// TwinCAT 3 PLC project PLC
// ProgramVersion: 3.1.4026.19
// libraries:
//   SPT Base Types, * (Beckhoff Automation LLC)
//   SPT Components, * (Beckhoff Automation LLC)
//   SPT Diagnostic, * (Beckhoff Automation LLC)
//   SPT EtherCat, * (Beckhoff Automation LLC)
//   SPT Event Logger, * (Beckhoff Automation LLC)
//   SPT Motion Control, * (Beckhoff Automation LLC)
//   SPT Utilities, * (Beckhoff Automation LLC)
//   Tc2_MC2, * (Beckhoff Automation GmbH)
//   Tc2_Standard, * (Beckhoff Automation GmbH)
//   Tc2_System, * (Beckhoff Automation GmbH)
//   Tc3_EventLogger, * (Beckhoff Automation GmbH)
//   Tc3_Module, * (Beckhoff Automation GmbH)
//   Tc3_PackML_V3, * (Beckhoff Automation GmbH)
// project tree:
//   / GlobalTextList.TcGTLO, PlcTask.TcTTO, Visualization Manager.TcVMO (not stored)
//   POUs/ MAIN.TcPOU
//   POUs/Modules/00 Machine/ Machine.TcPOU
//   POUs/Modules/01 Virtual Master/ VirtualMaster.TcPOU
//   POUs/Modules/02 Unwind/ Unwind.TcPOU
//   POUs/Modules/03 Draw/ DrawAxis.TcPOU
//   VISUs/ Visualization.TcVIS
// real-time tasks:
//   TASK PlcTask: cycle T#10ms, priority 20, ADS port 350
// motion (NC):
//   TASK NC-Task 1 SAF: cycle T#2ms, priority 4, ADS port 501
//   TASK NC-Task 1 SVB: cycle T#10ms, priority 8, ADS port 511
//   AXIS Virtual Master (id 1)
//   AXIS Unwind (id 2)
//   AXIS Draw (id 3)
// variable links:
//   PLC/PLC Instance <-> NC-Task 1 SAF/Axes/Draw
//     PlcTask Inputs/MAIN.Machine.Draw.Axis.BasicSlaveAxis._Axis.NcToPlc <-> Outputs/ToPlc
//     PlcTask Outputs/MAIN.Machine.Draw.Axis.BasicSlaveAxis._Axis.PlcToNc <-> Inputs/FromPlc
//   PLC/PLC Instance <-> NC-Task 1 SAF/Axes/Unwind
//     PlcTask Inputs/MAIN.Machine.Unwind.Axis.BasicSlaveAxis._Axis.NcToPlc <-> Outputs/ToPlc
//     PlcTask Outputs/MAIN.Machine.Unwind.Axis.BasicSlaveAxis._Axis.PlcToNc <-> Inputs/FromPlc
//   PLC/PLC Instance <-> NC-Task 1 SAF/Axes/Virtual Master
//     PlcTask Inputs/MAIN.Machine.VirtualMaster.Axis.BasicSlaveAxis._Axis.NcToPlc <-> Outputs/ToPlc
//     PlcTask Outputs/MAIN.Machine.VirtualMaster.Axis.BasicSlaveAxis._Axis.PlcToNc <-> Inputs/FromPlc

CONFIGURATION PLC
    RESOURCE PLC ON TwinCAT3
        TASK PlcTask(INTERVAL := T#10ms, PRIORITY := 20);
        PROGRAM MAIN WITH PlcTask : MAIN;
    END_RESOURCE
END_CONFIGURATION

// ---- POUs/MAIN.TcPOU
PROGRAM MAIN
VAR
	Machine : Machine := (Name := 'Machine');
END_VAR

(*All sample code provided by Beckhoff Automation LLC are for illustrative purposes only and are provided “as is” and without any warranties, express or implied. Actual implementations in applications will vary significantly. Beckhoff Automation LLC shall have no liability for, and does not waive any rights in relation to, any code samples that it provides or the use of such code samples for any purpose.*)

(*
	This code is not a full implementation as there is no use of MC_Reset or other needed code for actual machine use.
	Take note of step 10 in FB_Machine.Initialize, this is where the Axes are assigned to their Master.
	The Unwind Axis makes use of a Gear Ratio in its Coupling.
	There is no code to move the master axis, but it can be jogged from the NC for testing.
*)

// For Debug Only
_AppInfo.KeepOutputsOnBP := TRUE;

//
Machine.CyclicLogic();

END_PROGRAM

// ---- POUs/Modules/00 Machine/Machine.TcPOU
FUNCTION_BLOCK Machine EXTENDS FB_PackML_BaseModule
VAR
	VirtualMaster : VirtualMaster := (Name := 'Virtual Master');
	Unwind		  : Unwind		  := (Name := 'Unwind');
	Draw		  : DrawAxis	  := (Name := 'Draw');
END_VAR

METHOD PUBLIC CyclicLogic
IF NOT _InitComplete THEN
	_InitComplete := Initialize();
	RETURN;
END_IF

SUPER^.CyclicLogic();
END_METHOD

// Automatically enables and disables HMI control based on the PackML mode
METHOD PROTECTED HMIPermissions

// This method is called cyclically by CyclicLogic()
AllowHMIControl(ThisModuleOnly := TRUE);
END_METHOD

METHOD PROTECTED Initialize : BOOL;
Initialize := FALSE;
CASE DescendantSequenceState OF
	0: // Register Submodules
		RegisterSubmodule(VirtualMaster);
		RegisterSubmodule(Unwind);
		RegisterSubmodule(Draw);
		DescendantSequenceState := DescendantSequenceState + 10;

	10: // Assign axis references between Equipment Modules
		Unwind.MasterAxisRef	REF= VirtualMaster.AxisRef;
		Draw.MasterAxisRef		REF= VirtualMaster.AxisRef;
		DescendantSequenceState := DescendantSequenceState + 10;

	20:
		IF SUPER^.Initialize() THEN
			DescendantSequenceState := DescendantSequenceState + 10;
		END_IF

	30:
		Initialize := TRUE;
END_CASE
END_METHOD

END_FUNCTION_BLOCK

// ---- POUs/Modules/01 Virtual Master/VirtualMaster.TcPOU
FUNCTION_BLOCK VirtualMaster EXTENDS FB_PackML_BaseModule
VAR
	Axis : FB_Component_BasicSlaveAxis := (Name := 'Virtual Master Axis');
END_VAR

METHOD PROTECTED Aborting
//Mode is ignored
CASE SequenceState OF
	0:
		// Stop Axis
		Axis.Override := 100;
		IF Axis.Stop() OR Axis.Error THEN // This will also GearOut
			SequenceState := SequenceState + 10;
		END_IF

	10:
		IF Axis.Stopped THEN
			SequenceState := SequenceState + 10;
		END_IF

	20: // Disable Axis
		IF Axis.Disable() THEN
			SequenceState := SequenceState + 10;
		END_IF

	30:
		IF NOT Axis.Enabled THEN
			SequenceState := SequenceState + 10;
		END_IF

	40:
		SUPER^.Aborting();
END_CASE
END_METHOD

PROPERTY AxisRef : REFERENCE TO AXIS_REF
GET
AxisRef REF= Axis.Axis;
END_GET
END_PROPERTY

METHOD PROTECTED Completing
CASE _CurrentMode OF
	E_PMLUnitMode.Production:
		CASE SequenceState OF
			0:
				NoStateTasksToComplete := FALSE;
				IF Axis.Stop() THEN
					SequenceState := SequenceState + 10;
				END_IF

			10:
				IF Axis.Stopped THEN
					SequenceState := SequenceState + 10;
				END_IF

			20:
				StateTasksComplete := TRUE;
		END_CASE

	E_PMLUnitMode.Maintenance, E_PMLUnitMode.Manual:
		;
END_CASE

SUPER^.Completing();
END_METHOD

METHOD PUBLIC CyclicLogic
IF NOT _InitComplete THEN
	_InitComplete := Initialize();
	RETURN;
END_IF

SUPER^.CyclicLogic();
END_METHOD

METHOD PROTECTED Initialize : BOOL;
Initialize := FALSE;
CASE DescendantSequenceState OF
	0:
		RegisterComponent(Axis);
		DescendantSequenceState := DescendantSequenceState + 10;

	10:
		IF SUPER^.Initialize() THEN
			DescendantSequenceState := DescendantSequenceState + 10;
		END_IF

	20:
		Initialize := TRUE;
END_CASE
END_METHOD

METHOD PROTECTED Starting
CASE _CommandedMode OF
	E_PMLUnitMode.Production:
		CASE SequenceState OF
			0:
				NoStateTasksToComplete := FALSE;
				IF Axis.Enable() THEN
					SequenceState := SequenceState + 10;
				END_IF

			10:
				IF Axis.Enabled THEN
					SequenceState := SequenceState + 10;
				END_IF

			20:
				StateTasksComplete := TRUE;
		END_CASE
END_CASE

SUPER^.Starting();
END_METHOD

METHOD PROTECTED Stopping
CASE _CurrentMode OF
	E_PMLUnitMode.Production:
		CASE SequenceState OF
			0:
				NoStateTasksToComplete := FALSE;
				IF Axis.Stop() THEN //This will also GearOut
					SequenceState := SequenceState + 10;
				END_IF

			10:
				IF Axis.Stopped THEN
					SequenceState := SequenceState + 10;
				END_IF

			20:
				StateTasksComplete := TRUE;
		END_CASE
END_CASE

SUPER^.Stopping();
END_METHOD

END_FUNCTION_BLOCK

// ---- POUs/Modules/02 Unwind/Unwind.TcPOU
FUNCTION_BLOCK Unwind EXTENDS FB_PackML_BaseModule
VAR
	Axis	   : FB_Component_BasicSlaveAxis := (Name := 'Unwind Axis');
	_MasterRef : REFERENCE TO AXIS_REF;
END_VAR

METHOD PROTECTED Aborting
//Mode is ignored
CASE SequenceState OF
	0:
		NoStateTasksToComplete := FALSE;

		// Stop Axis
		Axis.Override := 100;
		IF Axis.Stop() OR Axis.Error THEN //This will also GearOut
			SequenceState := SequenceState + 10;
		END_IF

	10:
		IF Axis.Stopped THEN
			SequenceState := SequenceState + 10;
		END_IF

	20: // Disable Axis 
		IF Axis.Disable() THEN
			SequenceState := SequenceState + 10;
		END_IF

	30:
		IF NOT Axis.Enabled THEN
			SequenceState := SequenceState + 10;
		END_IF

	40:
		StateTasksComplete := TRUE;
END_CASE

SUPER^.Aborting();
END_METHOD

PROPERTY AxisRef : REFERENCE TO AXIS_REF
GET
AxisRef REF= Axis.Axis;
END_GET
END_PROPERTY

METHOD PROTECTED Completing
VAR_INST
	StopAxis : BOOL;
END_VAR
CASE _CurrentMode OF
	E_PMLUnitMode.Production:
		CASE SequenceState OF
			0:
				NoStateTasksToComplete := FALSE;
				IF Axis.InGear AND_THEN Axis.Master1.Status.StandStill THEN //Wait for Master Axis to Stop
					StopAxis := TRUE;
				ELSIF NOT Axis.InGear THEN
					StopAxis := TRUE;
				ELSE
					StopAxis := FALSE;
				END_IF

				IF StopAxis AND_THEN Axis.Stop() THEN // This will also GearOut
					SequenceState := SequenceState + 10;
				END_IF

			10:
				IF Axis.Stopped THEN
					SequenceState := SequenceState + 10;
				END_IF

			20:
				StateTasksComplete := TRUE;
		END_CASE

	E_PMLUnitMode.Maintenance, E_PMLUnitMode.Manual:
		;
END_CASE

SUPER^.Completing();
END_METHOD

METHOD PUBLIC CyclicLogic
IF NOT _InitComplete THEN
	_InitComplete := Initialize();
	RETURN;
END_IF

SUPER^.CyclicLogic();
END_METHOD

METHOD PROTECTED Initialize : BOOL;
Initialize := FALSE;
CASE DescendantSequenceState OF
	0:
		RegisterComponent(Axis);
		DescendantSequenceState := DescendantSequenceState + 10;

	10:
		IF SUPER^.Initialize() THEN
			DescendantSequenceState := DescendantSequenceState + 10;
		END_IF

	20:
		Initialize := TRUE;
END_CASE
END_METHOD

PROPERTY MasterAxisRef : REFERENCE TO AXIS_REF
SET
IF __ISVALIDREF(MasterAxisRef) THEN
	_MasterRef REF= MasterAxisRef;
END_IF
END_SET
END_PROPERTY

METHOD PROTECTED Starting
CASE _CommandedMode OF
	E_PMLUnitMode.Production:
		CASE SequenceState OF
			0:
				NoStateTasksToComplete := FALSE;
				IF Axis.Enable() THEN
					SequenceState := SequenceState + 10;
				END_IF

			10:
				IF Axis.Enabled THEN
					SequenceState := SequenceState + 10;
				END_IF

			20:
				Axis.Master1	  REF= _MasterRef;
				Axis.RatioMaster1 := 0.5; //Can be set at anytime and changed while in motion
				IF Axis.GearIn() THEN
					SequenceState := SequenceState + 10;
				END_IF

			30:
				IF Axis.InGear THEN
					SequenceState := SequenceState + 10;
				END_IF

			40:
				StateTasksComplete := TRUE;
		END_CASE
END_CASE

SUPER^.Starting();
END_METHOD

METHOD PROTECTED Stopping
CASE _CurrentMode OF
	E_PMLUnitMode.Production:
		CASE SequenceState OF
			0:
				NoStateTasksToComplete := FALSE;
				IF Axis.Stop() THEN //This will also GearOut
					SequenceState := SequenceState + 10;
				END_IF

			10:
				IF Axis.Stopped THEN
					SequenceState := SequenceState + 10;
				END_IF

			20:
				StateTasksComplete := TRUE;
		END_CASE
END_CASE

SUPER^.Stopping();
END_METHOD

END_FUNCTION_BLOCK

// ---- POUs/Modules/03 Draw/DrawAxis.TcPOU
FUNCTION_BLOCK DrawAxis EXTENDS FB_PackML_BaseModule
VAR
	Axis	   : FB_Component_BasicSlaveAxis := (Name := 'Draw Axis');
	_MasterRef : REFERENCE TO AXIS_REF;
END_VAR

METHOD PROTECTED Aborting
//Mode is ignored
CASE SequenceState OF
	0:
		NoStateTasksToComplete := FALSE;

		// Stop Axis
		Axis.Override := 100;
		IF Axis.Stop() OR Axis.Error THEN //This will also GearOut
			SequenceState := SequenceState + 10;
		END_IF

	10:
		IF Axis.Stopped THEN
			SequenceState := SequenceState + 10;
		END_IF

	20: // Disable Axis
		IF Axis.Disable() THEN
			SequenceState := SequenceState + 10;
		END_IF

	30:
		IF NOT Axis.Enabled THEN
			SequenceState := SequenceState + 10;
		END_IF

	40:
		StateTasksComplete := TRUE;
END_CASE

SUPER^.Aborting();
END_METHOD

PROPERTY AxisRef : REFERENCE TO AXIS_REF
GET
AxisRef REF= Axis.Axis;
END_GET
END_PROPERTY

METHOD PROTECTED Completing
VAR_INST
	StopAxis : BOOL;
END_VAR
CASE _CurrentMode OF
	E_PMLUnitMode.Production:
		CASE SequenceState OF
			0:
				NoStateTasksToComplete := FALSE;
				IF Axis.InGear AND_THEN Axis.Master1.Status.StandStill THEN //Wait for Master Axis to Stop
					StopAxis := TRUE;
				ELSIF NOT Axis.InGear THEN
					StopAxis := TRUE;
				ELSE
					StopAxis := FALSE;
				END_IF

				IF StopAxis AND_THEN Axis.Stop() THEN // This will also GearOut
					SequenceState := SequenceState + 10;
				END_IF

			10:
				IF Axis.Stopped THEN
					SequenceState := SequenceState + 10;
				END_IF

			20:
				StateTasksComplete := TRUE;
		END_CASE

	E_PMLUnitMode.Maintenance, E_PMLUnitMode.Manual:
		;
END_CASE

SUPER^.Completing();
END_METHOD

METHOD PUBLIC CyclicLogic
IF NOT _InitComplete THEN
	_InitComplete := Initialize();
	RETURN;
END_IF

SUPER^.CyclicLogic();
END_METHOD

METHOD PROTECTED Initialize : BOOL;
Initialize := FALSE;
CASE DescendantSequenceState OF
	0:
		RegisterComponent(Axis);
		DescendantSequenceState := DescendantSequenceState + 10;

	10:
		IF SUPER^.Initialize() THEN
			DescendantSequenceState := DescendantSequenceState + 10;
		END_IF

	20:
		Initialize := TRUE;
END_CASE
END_METHOD

PROPERTY MasterAxisRef : REFERENCE TO AXIS_REF
SET
IF __ISVALIDREF(MasterAxisRef) THEN
	_MasterRef REF= MasterAxisRef;
END_IF
END_SET
END_PROPERTY

METHOD PROTECTED Starting
CASE _CommandedMode OF
	E_PMLUnitMode.Production:
		CASE SequenceState OF
			0:
				NoStateTasksToComplete := FALSE;
				IF Axis.Enable() THEN
					SequenceState := SequenceState + 10;
				END_IF

			10:
				IF Axis.Enabled THEN
					SequenceState := SequenceState + 10;
				END_IF

			20:
				Axis.Master1 REF= _MasterRef;
				IF Axis.GearIn() THEN
					SequenceState := SequenceState + 10;
				END_IF

			30:
				IF Axis.InGear THEN
					SequenceState := SequenceState + 10;
				END_IF

			40:
				StateTasksComplete := TRUE;
		END_CASE
END_CASE

SUPER^.Starting();
END_METHOD

METHOD PROTECTED Stopping
CASE _CurrentMode OF
	E_PMLUnitMode.Production:
		CASE SequenceState OF
			0:
				NoStateTasksToComplete := FALSE;
				IF Axis.Stop() THEN //This will also GearOut
					SequenceState := SequenceState + 10;
				END_IF

			10:
				IF Axis.Stopped THEN
					SequenceState := SequenceState + 10;
				END_IF

			20:
				StateTasksComplete := TRUE;
		END_CASE
END_CASE

SUPER^.Stopping();
END_METHOD

END_FUNCTION_BLOCK

// ---- VISUs/Visualization.TcVIS
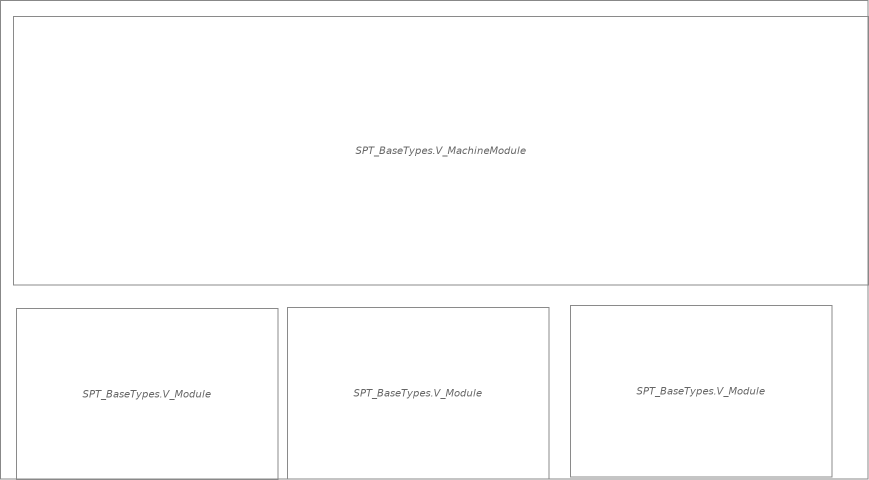
VISUALIZATION Visualization  // 869x480
    Frame (13,16 856x269)
        shows SPT_BaseTypes.V_MachineModule(HMI := MAIN.Machine.PackMLBaseModule_HMI)
    Frame (16,308 262x172)
        shows SPT_BaseTypes.V_Module(HMI := MAIN.Machine.Draw.PackMLBaseModule_HMI)
    Frame (287,307 262x172)
        shows SPT_BaseTypes.V_Module(HMI := MAIN.Machine.Unwind.PackMLBaseModule_HMI)
    Frame (570,305 262x172)
        shows SPT_BaseTypes.V_Module(HMI := MAIN.Machine.VirtualMaster.PackMLBaseModule_HMI)
END_VISUALIZATION
